(* Schneider Machine Expert - Basic project Tank_Level_v19, file version 3.0.0.0 *)
(* ProjectInformations: Name=New project *)

HARDWARE
  Cpu 0: TM221CE16T
  ModuleExtensionObject 0: TM3AI4/G
  EthernetConfiguration: NetworkName=M221, IpAllocationMode=FixedAddress, IpAddress=0.0.0.0, SubnetMask=0.0.0.0
  SerialLineConfiguration: Baud=Baud19200, Parity=ParityEven, DataBits=DataBits8, StopBits=StopBits1, PhysicalMedium=PhysicalMediumRs485, TransmissionMode=TransmissionModeModbusRtu, SlaveId=1, Addressing=SlaveAddressing
  MastTask: UsePeriodScanMode=false, PeriodScan=100
  FastTask: Period=255
  CpuBehavior: StartingMode=StartAsPreviousState, AutoSaveRamOnEeprom=true, WatchdogPeriod=250

SYMBOLS  (address, symbol, comment, settings)
  %M0       ENABLE_OPERATION
  %M1       TANK_LEVEL_LOW
  %M2       TANK_LEVEL_HIGH
  %Q0.0     INLET_VALVE
  %Q0.1     OUTLET_VALVE
  %IW1.0    TANK_LEVEL  [Type=Type_4_20mA, Scope=Scope_Customized, Minimum=300, Maximum=3000]

POU New POU
  (* SectionNumber=0 *)

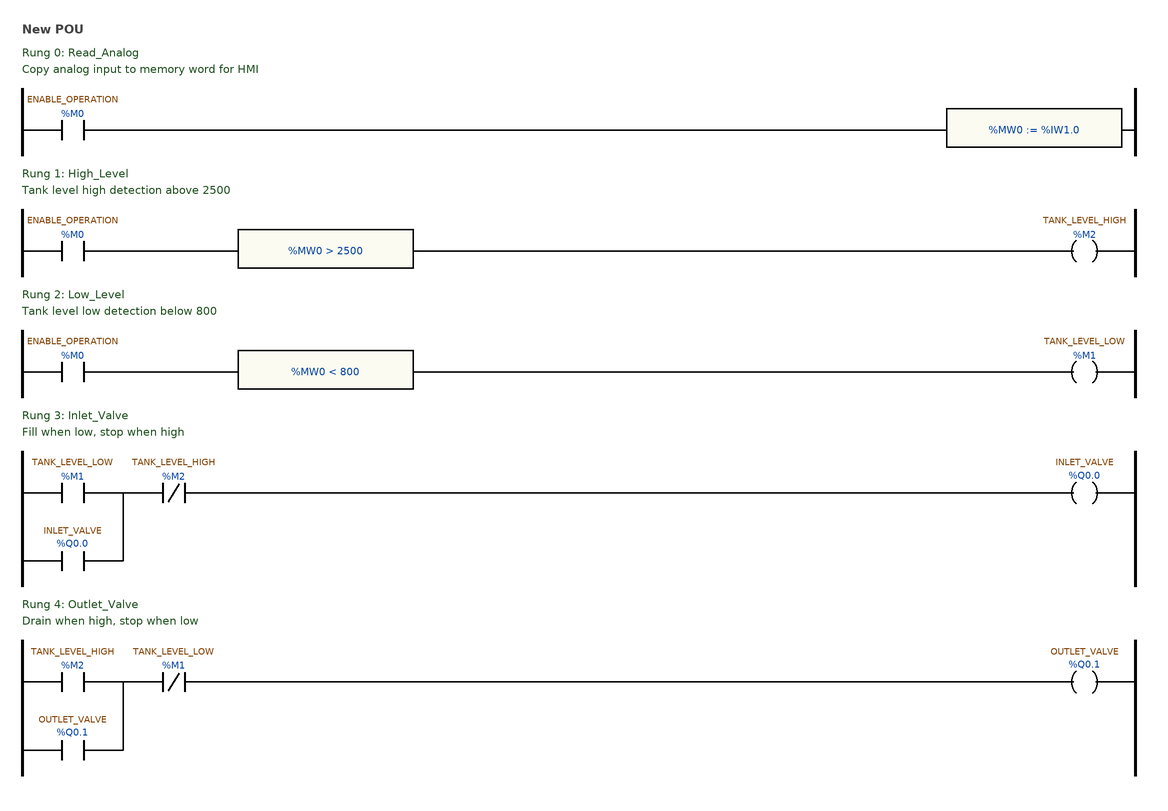

// Rung 0: Read_Analog
// Copy analog input to memory word for HMI
  LD %M0                  (* ENABLE_OPERATION *)
  [ %MW0 := %IW1.0 ]      (* TANK_LEVEL *)
  // as ST:
  //   IF ENABLE_OPERATION THEN %MW0 := TANK_LEVEL; END_IF;

// Rung 1: High_Level
// Tank level high detection above 2500
  LD %M0                  (* ENABLE_OPERATION *)
  AND [ %MW0 > 2500 ]
  ST %M2                  (* TANK_LEVEL_HIGH *)
  // as ST:
  //   TANK_LEVEL_HIGH := ENABLE_OPERATION AND %MW0 > 2500;

// Rung 2: Low_Level
// Tank level low detection below 800
  LD %M0                  (* ENABLE_OPERATION *)
  AND [ %MW0 < 800 ]
  ST %M1                  (* TANK_LEVEL_LOW *)
  // as ST:
  //   TANK_LEVEL_LOW := ENABLE_OPERATION AND %MW0 < 800;

// Rung 3: Inlet_Valve
// Fill when low, stop when high
  LD %M1                  (* TANK_LEVEL_LOW *)
  OR %Q0.0                (* INLET_VALVE *)
  ANDN %M2                (* TANK_LEVEL_HIGH *)
  ST %Q0.0                (* INLET_VALVE *)
  // as ST:
  //   INLET_VALVE := (TANK_LEVEL_LOW OR INLET_VALVE) AND NOT TANK_LEVEL_HIGH;

// Rung 4: Outlet_Valve
// Drain when high, stop when low
  LD %M2                  (* TANK_LEVEL_HIGH *)
  OR %Q0.1                (* OUTLET_VALVE *)
  ANDN %M1                (* TANK_LEVEL_LOW *)
  ST %Q0.1                (* OUTLET_VALVE *)
  // as ST:
  //   OUTLET_VALVE := (TANK_LEVEL_HIGH OR OUTLET_VALVE) AND NOT TANK_LEVEL_LOW;
